(* PLC project Unnamed, Unknown Unnamed 1 *)
(* stored: creationDateTime 2026-03-03T10:17:37, modificationDateTime 2026-03-03T10:36:34 *)

PROGRAM program0
  VAR
    Cycle_Complete AT %IX0.1 : BOOL;
    Service_Due AT %M05 : BOOL;
    Reset AT %IX0.2 : BOOL;
  END_VAR
  VAR
    Program_Value : INT := 100;
    CTU0 : CTU;
  END_VAR
  VAR  (* added by the conversion: wires and edge detectors of the diagram *)
    F_TRIG1 : F_TRIG;
    R_TRIG2 : R_TRIG;
  END_VAR

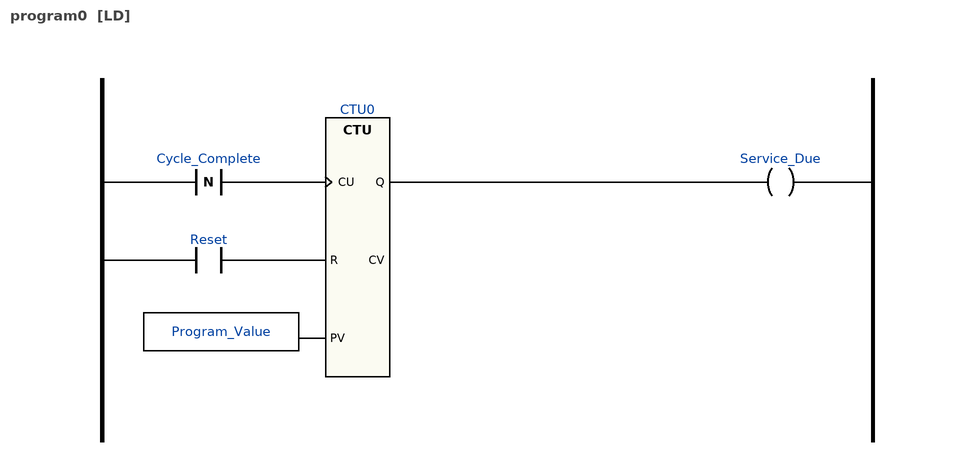
(* LD diagram, written out as Structured Text *)
F_TRIG1(CLK := Cycle_Complete);
R_TRIG2(CLK := F_TRIG1.Q);
CTU0(CU := R_TRIG2.Q, R := Reset, PV := Program_Value);
Service_Due := CTU0.Q;
END_PROGRAM

CONFIGURATION Config0
  RESOURCE Res0 ON PLC
    TASK task0(INTERVAL := T#20ms, PRIORITY := 0);
    PROGRAM instance0 WITH task0 : program0;
  END_RESOURCE
END_CONFIGURATION
